(* IEC 61131-3 sources: AXOpen/src/data/tests/AXOpen.Data.Tests_L1/ax/src/StationData, 2 files *)

(* ---- StationData.st ---- *)
USING AXOpen.Core;
USING AXOpen.Data;

NAMESPACE Tests_L1

    {S7.extern=ReadWrite}
    CLASS PUBLIC StationData EXTENDS AXOpen.Data.AxoDataEntity
        VAR PUBLIC
            //StationPass : BOOL;
            CounterDelay : ULINT;
        END_VAR
    END_CLASS

END_NAMESPACE

(* ---- StationDataManager.st ---- *)
USING AXOpen.Core;
USING AXOpen.Data;

NAMESPACE Tests_L1

    {S7.extern=ReadWrite}
    CLASS PUBLIC StationDataManager EXTENDS AXOpen.Data.AxoDataExchange
        VAR PUBLIC
            {#ix-generic:TOnline}
            {#ix-generic:TPlain as POCO}
            {#ix-attr:[AXOpen.Data.AxoDataEntityAttribute]}
            Set : Tests_L1.StationData;
        END_VAR
    END_CLASS

END_NAMESPACE
